PROGRAM PRGTEST
VAR
	sequencer_test : FB_Sequencer_Test;
	step_manager_test : FB_StepManagerBasic_Test;
END_VAR

TcUnit.RUN();

END_PROGRAM

(* stored: Version 1.1.0.1, ProductVersion 3.1.4024.12
   POU PRGTEST: Id {cb0dada2-790f-48b3-8702-fc17bd7e66f5}, SpecialFunc None *)
